PROGRAM StateMachine
VAR
	tolerance:UINT:=20;
	RS_Idle: RS;
	RS_Homing: RS;
	RS_place:RS;
	RS_Pick:RS;
	SR_ESTOP:SR;
	
	bValveClosed: BOOL;
	bValveOpen: BOOL;
	
	HorizontalState: AboutEqual;
	VerticalState: AboutEqual;
	RotationState: AboutEqual;
	bStateIdle: BOOL;
	bStateHoming: BOOL;
	bStatePick: BOOL;
	bStatePlace: BOOL;
	bStateEStop: BOOL;
	//check if position has reached
	Horizontal_Pick: BOOL;
	Vertical_Pick: BOOL;
	Rotation_Pick: BOOL;
	Horizontal_Place: BOOL;
	Vertical_Place: BOOL;
	Rotation_Place: BOOL;
	HorizontalState_b: AboutEqual;
	VerticalState_b: AboutEqual;
	RotationState_b: AboutEqual;
	HorizontalState_a: AboutEqual;
	VerticalState_a: AboutEqual;
	RotationState_a: AboutEqual;
END_VAR
VAR // added by the converter: edge detectors and wires of the graphical bodies
    _w1, _w2, _w3 : BOOL;
END_VAR

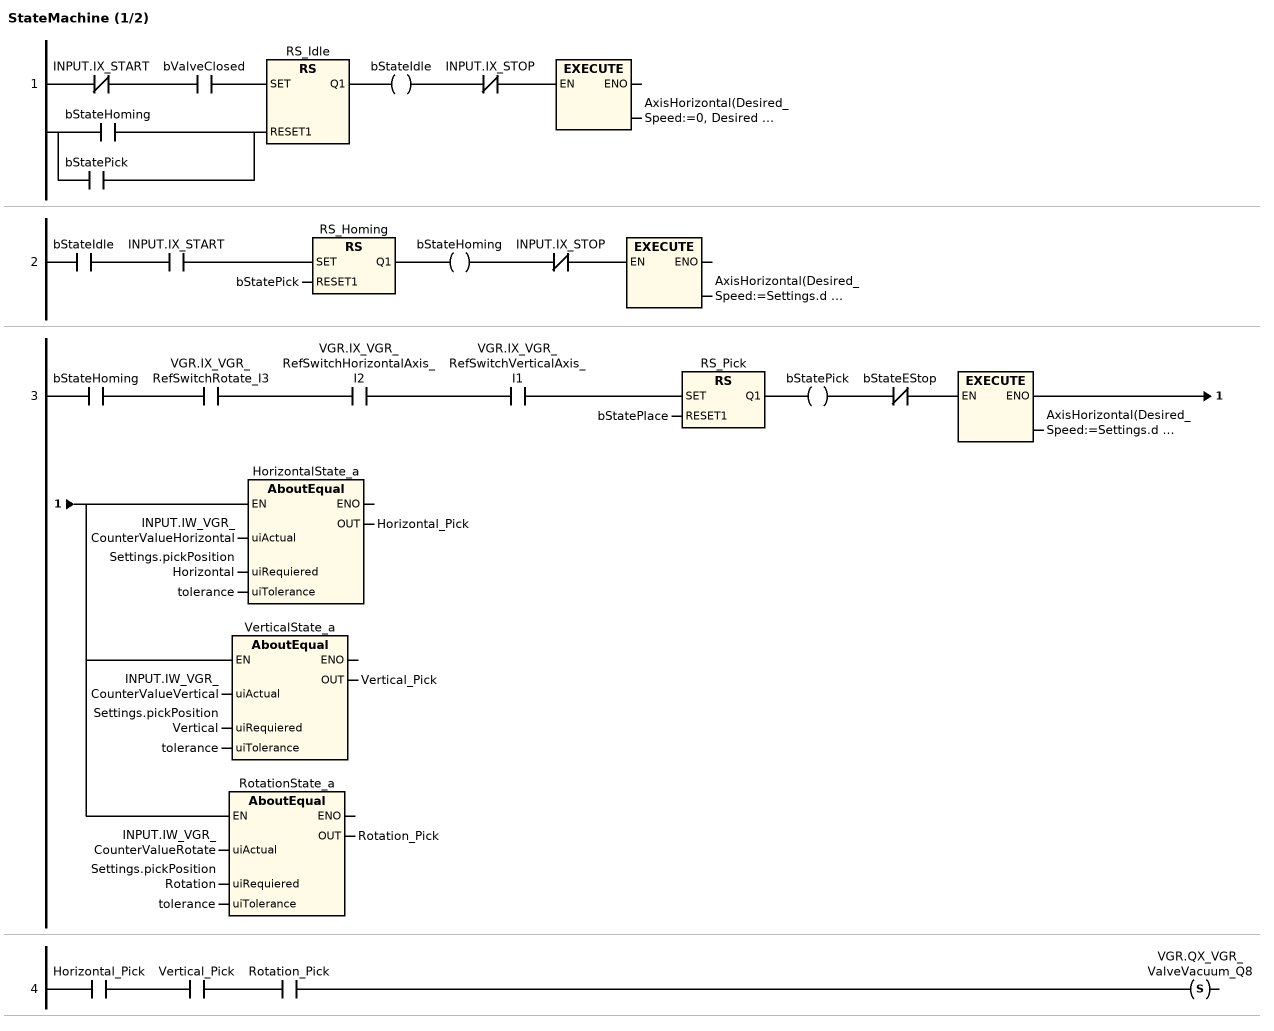
// NETWORK 1
RS_Idle(SET := NOT INPUT.IX_START AND bValveClosed, RESET1 := bStateHoming OR bStatePick); // RS
bStateIdle := RS_Idle.Q1;
IF RS_Idle.Q1 AND NOT INPUT.IX_STOP THEN
    AxisHorizontal(Desired_Speed:=0, Desired_Position:= input.IW_VGR_CounterValueHorizontal, tolerance:=20);
    AxisVertical(Desired_Speed:=0,
    			Desired_Position:= input.IW_VGR_CounterValueVertical,
    			tolerance:=20);
    AxisRotate(Desired_Speed:=0,
    			Desired_Position:= input.IW_VGR_CounterValueRotate,
    			tolerance:=20);
    Settings.CurrentState:='IDLE';
END_IF

// NETWORK 2
RS_Homing(SET := bStateIdle AND INPUT.IX_START, RESET1 := bStatePick); // RS
bStateHoming := RS_Homing.Q1;
IF RS_Homing.Q1 AND NOT INPUT.IX_STOP THEN
    AxisHorizontal(Desired_Speed:=Settings.desiredSpeedHorizontal,
    			Desired_Position:= 0,
    			tolerance:=tolerance);
    AxisVertical(Desired_Speed:=Settings.desiredSpeedVertical,
    			Desired_Position:= 0,
    			tolerance:=tolerance);
    AxisRotate(Desired_Speed:= Settings.desiredSpeedRotation,
    			Desired_Position:= 0,
    			tolerance:=tolerance);
    Settings.CurrentState:="HOME";
END_IF

// NETWORK 3
RS_Pick(SET := bStateHoming AND VGR.IX_VGR_RefSwitchRotate_I3 AND VGR.IX_VGR_RefSwitchHorizontalAxis_I2 AND VGR.IX_VGR_RefSwitchVerticalAxis_I1, RESET1 := bStatePlace); // RS
bStatePick := RS_Pick.Q1;
_w1 := RS_Pick.Q1 AND NOT bStateEStop;
IF _w1 THEN
    AxisHorizontal(Desired_Speed:=Settings.desiredSpeedHorizontal,
    			Desired_Position:= settings.pickPositionHorizontal,
    			tolerance:=tolerance);
    AxisVertical(Desired_Speed:=Settings.desiredSpeedVertical,
    			Desired_Position:= Settings.pickPositionVertical,
    			tolerance:=tolerance);
    AxisRotate(Desired_Speed:= Settings.desiredSpeedRotation,
    			Desired_Position:= settings.pickPositionRotation,
    			tolerance:=tolerance);
    Settings.CurrentState:='PICK';
END_IF
IF _w1 THEN
    HorizontalState_a(
        uiActual := INPUT.IW_VGR_CounterValueHorizontal,
        uiRequiered := Settings.pickPositionHorizontal,
        uiTolerance := tolerance,
        OUT => Horizontal_Pick); // AboutEqual
END_IF
IF _w1 THEN
    VerticalState_a(
        uiActual := INPUT.IW_VGR_CounterValueVertical,
        uiRequiered := Settings.pickPositionVertical,
        uiTolerance := tolerance,
        OUT => Vertical_Pick); // AboutEqual
END_IF
IF _w1 THEN
    RotationState_a(
        uiActual := INPUT.IW_VGR_CounterValueRotate,
        uiRequiered := Settings.pickPositionRotation,
        uiTolerance := tolerance,
        OUT => Rotation_Pick); // AboutEqual
END_IF

// NETWORK 4
VGR.QX_VGR_ValveVacuum_Q8 S= Horizontal_Pick AND Vertical_Pick AND Rotation_Pick;

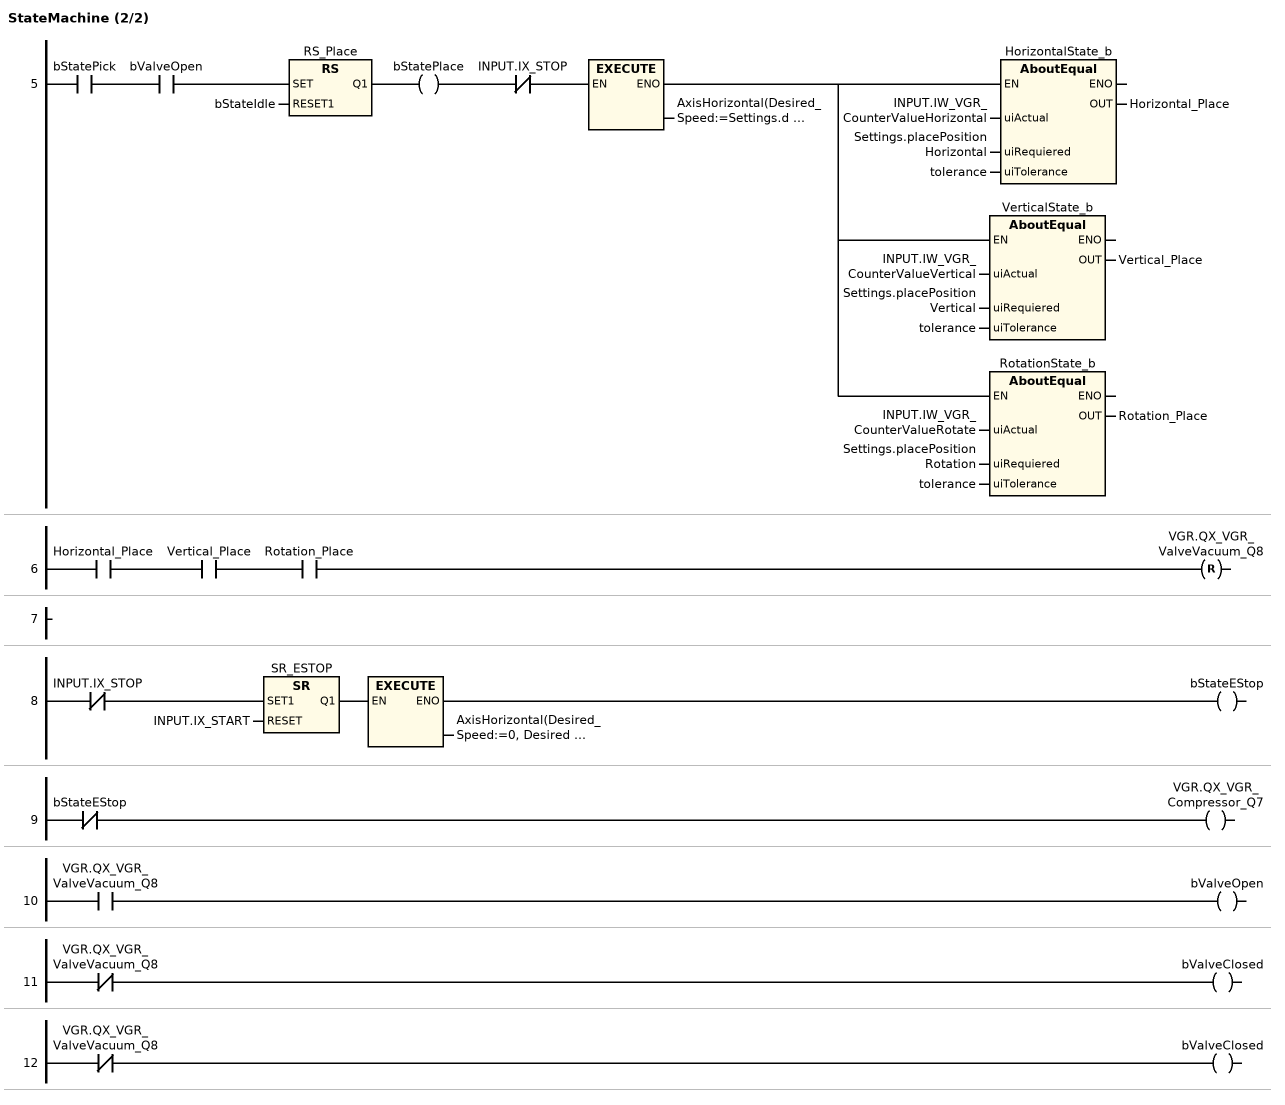
// NETWORK 5
RS_Place(SET := bStatePick AND bValveOpen, RESET1 := bStateIdle); // RS
bStatePlace := RS_Place.Q1;
_w2 := RS_Place.Q1 AND NOT INPUT.IX_STOP;
IF _w2 THEN
    AxisHorizontal(Desired_Speed:=Settings.desiredSpeedHorizontal,
    			Desired_Position:= Settings.placePositionHorizontal,
    			tolerance:=20);
    AxisVertical(Desired_Speed:=Settings.desiredSpeedVertical,
    			 Desired_Position:= Settings.placePositionVertical,
    	   		 tolerance:=20);
    AxisRotate(Desired_Speed:=Settings.desiredSpeedRotation,
    			Desired_Position:= Settings.placePositionRotation,
    			tolerance:=20);
    Settings.CurrentState:='PLACE';
END_IF
IF _w2 THEN
    HorizontalState_b(
        uiActual := INPUT.IW_VGR_CounterValueHorizontal,
        uiRequiered := Settings.placePositionHorizontal,
        uiTolerance := tolerance,
        OUT => Horizontal_Place); // AboutEqual
END_IF
IF _w2 THEN
    VerticalState_b(
        uiActual := INPUT.IW_VGR_CounterValueVertical,
        uiRequiered := Settings.placePositionVertical,
        uiTolerance := tolerance,
        OUT => Vertical_Place); // AboutEqual
END_IF
IF _w2 THEN
    RotationState_b(
        uiActual := INPUT.IW_VGR_CounterValueRotate,
        uiRequiered := Settings.placePositionRotation,
        uiTolerance := tolerance,
        OUT => Rotation_Place); // AboutEqual
END_IF

// NETWORK 6
VGR.QX_VGR_ValveVacuum_Q8 R= Horizontal_Place AND Vertical_Place AND Rotation_Place;

// NETWORK 7

// NETWORK 8
SR_ESTOP(SET1 := NOT INPUT.IX_STOP, RESET := INPUT.IX_START); // SR
_w3 := SR_ESTOP.Q1;
IF _w3 THEN
    AxisHorizontal(Desired_Speed:=0, Desired_Position:= input.IW_VGR_CounterValueHorizontal, tolerance:=20);
    AxisVertical(Desired_Speed:=0,
    			Desired_Position:= input.IW_VGR_CounterValueVertical,
    			tolerance:=20);
    AxisRotate(Desired_Speed:=0,
    			Desired_Position:= input.IW_VGR_CounterValueRotate,
    			tolerance:=20);
    Settings.CurrentState:='E_STOP';
END_IF
bStateEStop := _w3;

// NETWORK 9
VGR.QX_VGR_Compressor_Q7 := NOT bStateEStop;

// NETWORK 10
bValveOpen := VGR.QX_VGR_ValveVacuum_Q8;

// NETWORK 11
bValveClosed := NOT VGR.QX_VGR_ValveVacuum_Q8;

// NETWORK 12
bValveClosed := NOT VGR.QX_VGR_ValveVacuum_Q8;

END_PROGRAM

(* stored: Version 1.1.0.1, ProductVersion 3.1.4024.12
   POU StateMachine: Id {102b109e-5d65-44f6-9162-be32ce46a64a}, SpecialFunc None *)
